// TwinCAT 3 PLC project PLC
// ProgramVersion: 3.1.4023.0
// libraries:
//   Tc2_EtherCAT, * (Beckhoff Automation GmbH)
//   Tc2_Standard, * (Beckhoff Automation GmbH)
//   Tc2_System, * (Beckhoff Automation GmbH)
//   Tc3_Module, * (Beckhoff Automation GmbH)
//   VisuDialogs, * (System)
// project tree:
//   / FastEL5131Task.TcTTO, GlobalTextList.TcGTLO, PlcTask.TcTTO, Visualization Manager.TcVMO (not stored)
//   POUs/ FB_PulseDiv.TcPOU, MAIN.TcPOU, MAINEL5131.TcPOU
//   VISUs/ MAINVISU.TcVIS
// real-time tasks:
//   TASK PlcTask: cycle T#10ms, priority 20, ADS port 350
//   TASK FastEL5131Task: cycle T#200us, priority 1, ADS port 351
// I/O:
//   DEVICE Device 1 (EtherCAT), AmsNetId 5.25.121.244.2.1
//     Term 1 (EK1100) [EK1100 EtherCAT Coupler (2A E-Bus)]
//       Term 2 (EL5131) [EL5131 1Ch. Inc. Encoder 5V (RS422,TTL), 2x24V DC Output]
//       Term 4 (EL5101) [EL5101 1Ch. Inc. Encoder 5V]
//       Term 3 (EL9011)
// variable links:
//   PLC Instance <-> Device 1 (EtherCAT)/Term 1 (EK1100)/Term 2 (EL5131)
//     FastEL5131Task Inputs/MAINEL5131.myPulseDiv.amsNetIdEL5131 <-> InfoData/AdsAddr/netId
//     FastEL5131Task Inputs/MAINEL5131.myPulseDiv.iEL5131CounterVal <-> ENC Status Channel 1/Counter value
//     FastEL5131Task Inputs/MAINEL5131.myPulseDiv.wPortEL5131 <-> InfoData/AdsAddr/port
//     FastEL5131Task Outputs/MAINEL5131.myPulseDiv.bEnbThreshOutputs <-> ENC Control Output Channel 1/Control Output/Control/Enable thresholds output
//     FastEL5131Task Outputs/MAINEL5131.myPulseDiv.bEnbThreshOutputs2 <-> ENC Control Output Channel 2/Control Output/Control/Enable thresholds output
//     FastEL5131Task Outputs/MAINEL5131.myPulseDiv.bForceResetCounter <-> ENC Control Channel 1/Control/Set counter
//     FastEL5131Task Outputs/MAINEL5131.myPulseDiv.bSetDigitalOut <-> ENC Control Output Channel 1/Control Output/Control/Set digital output
//     FastEL5131Task Outputs/MAINEL5131.myPulseDiv.bSetDigitalOut2 <-> ENC Control Output Channel 2/Control Output/Control/Set digital output
//     FastEL5131Task Outputs/MAINEL5131.myPulseDiv.iForceResetCntVal <-> ENC Control Channel 1/Set counter value
//     FastEL5131Task Outputs/MAINEL5131.myPulseDiv.iNbOfOutputEvents <-> ENC Control Output Channel 1/Control Output/Number of output events
//     FastEL5131Task Outputs/MAINEL5131.myPulseDiv.iOutStates_1[1] <-> ENC Control Output Channel 1/Control Output/Output state/Output state 1
//     FastEL5131Task Outputs/MAINEL5131.myPulseDiv.iOutStates_1[2] <-> ENC Control Output Channel 1/Control Output/Output state/Output state 2
//     FastEL5131Task Outputs/MAINEL5131.myPulseDiv.iOutStates_1[3] <-> ENC Control Output Channel 1/Control Output/Output state/Output state 3
//     FastEL5131Task Outputs/MAINEL5131.myPulseDiv.iOutStates_1[4] <-> ENC Control Output Channel 1/Control Output/Output state/Output state 4
//     FastEL5131Task Outputs/MAINEL5131.myPulseDiv.iOutStates_1[5] <-> ENC Control Output Channel 1/Control Output/Output state/Output state 5
//     FastEL5131Task Outputs/MAINEL5131.myPulseDiv.iOutStates_1[6] <-> ENC Control Output Channel 1/Control Output/Output state/Output state 6
//     FastEL5131Task Outputs/MAINEL5131.myPulseDiv.iOutStates_1[7] <-> ENC Control Output Channel 1/Control Output/Output state/Output state 7
//     FastEL5131Task Outputs/MAINEL5131.myPulseDiv.iOutStates_1[8] <-> ENC Control Output Channel 1/Control Output/Output state/Output state 8
//     FastEL5131Task Outputs/MAINEL5131.myPulseDiv.iOutStates_2[1] <-> ENC Control Output Channel 2/Control Output/Output state/Output state 1
//     FastEL5131Task Outputs/MAINEL5131.myPulseDiv.iOutStates_2[2] <-> ENC Control Output Channel 2/Control Output/Output state/Output state 2
//     FastEL5131Task Outputs/MAINEL5131.myPulseDiv.iOutStates_2[3] <-> ENC Control Output Channel 2/Control Output/Output state/Output state 3
//     FastEL5131Task Outputs/MAINEL5131.myPulseDiv.iOutStates_2[4] <-> ENC Control Output Channel 2/Control Output/Output state/Output state 4
//     FastEL5131Task Outputs/MAINEL5131.myPulseDiv.iOutStates_2[5] <-> ENC Control Output Channel 2/Control Output/Output state/Output state 5
//     FastEL5131Task Outputs/MAINEL5131.myPulseDiv.iOutStates_2[6] <-> ENC Control Output Channel 2/Control Output/Output state/Output state 6
//     FastEL5131Task Outputs/MAINEL5131.myPulseDiv.iOutStates_2[7] <-> ENC Control Output Channel 2/Control Output/Output state/Output state 7
//     FastEL5131Task Outputs/MAINEL5131.myPulseDiv.iOutStates_2[8] <-> ENC Control Output Channel 2/Control Output/Output state/Output state 8
//     FastEL5131Task Outputs/MAINEL5131.myPulseDiv.iThresholds_1 <-> ENC Control Output Channel 1/Control Output/Threshold/Threshold 1
//     FastEL5131Task Outputs/MAINEL5131.myPulseDiv.iThresholds_2 <-> ENC Control Output Channel 2/Control Output/Threshold/Threshold 1
//     FastEL5131Task Outputs/MAINEL5131.myPulseDiv.iThresholds_1 @bit 32 <-> ENC Control Output Channel 1/Control Output/Threshold/Threshold 2
//     FastEL5131Task Outputs/MAINEL5131.myPulseDiv.iThresholds_1 @bit 64 <-> ENC Control Output Channel 1/Control Output/Threshold/Threshold 3
//     FastEL5131Task Outputs/MAINEL5131.myPulseDiv.iThresholds_1 @bit 96 <-> ENC Control Output Channel 1/Control Output/Threshold/Threshold 4
//     FastEL5131Task Outputs/MAINEL5131.myPulseDiv.iThresholds_1 @bit 128 <-> ENC Control Output Channel 1/Control Output/Threshold/Threshold 5
//     FastEL5131Task Outputs/MAINEL5131.myPulseDiv.iThresholds_1 @bit 160 <-> ENC Control Output Channel 1/Control Output/Threshold/Threshold 6
//     FastEL5131Task Outputs/MAINEL5131.myPulseDiv.iThresholds_1 @bit 192 <-> ENC Control Output Channel 1/Control Output/Threshold/Threshold 7
//     FastEL5131Task Outputs/MAINEL5131.myPulseDiv.iThresholds_1 @bit 224 <-> ENC Control Output Channel 1/Control Output/Threshold/Threshold 8
//     FastEL5131Task Outputs/MAINEL5131.myPulseDiv.iThresholds_2 @bit 32 <-> ENC Control Output Channel 2/Control Output/Threshold/Threshold 2
//     FastEL5131Task Outputs/MAINEL5131.myPulseDiv.iThresholds_2 @bit 64 <-> ENC Control Output Channel 2/Control Output/Threshold/Threshold 3
//     FastEL5131Task Outputs/MAINEL5131.myPulseDiv.iThresholds_2 @bit 96 <-> ENC Control Output Channel 2/Control Output/Threshold/Threshold 4
//     FastEL5131Task Outputs/MAINEL5131.myPulseDiv.iThresholds_2 @bit 128 <-> ENC Control Output Channel 2/Control Output/Threshold/Threshold 5
//     FastEL5131Task Outputs/MAINEL5131.myPulseDiv.iThresholds_2 @bit 160 <-> ENC Control Output Channel 2/Control Output/Threshold/Threshold 6
//     FastEL5131Task Outputs/MAINEL5131.myPulseDiv.iThresholds_2 @bit 192 <-> ENC Control Output Channel 2/Control Output/Threshold/Threshold 7
//     FastEL5131Task Outputs/MAINEL5131.myPulseDiv.iThresholds_2 @bit 224 <-> ENC Control Output Channel 2/Control Output/Threshold/Threshold 8
//   PLC Instance <-> Device 1 (EtherCAT)/Term 1 (EK1100)/Term 4 (EL5101)
//     PlcTask Inputs/MAIN.iCounterValueDoubleCheckEL5101 <-> ENC Status/Counter value
//     PlcTask Outputs/MAIN.bResetCounterEL5101 <-> ENC Control/Control/Set counter
//     PlcTask Outputs/MAIN.iSetCounterValueEL5101ForReset <-> ENC Control/Set counter value

CONFIGURATION PLC
    RESOURCE PLC ON TwinCAT3
        TASK FastEL5131Task(INTERVAL := T#200us, PRIORITY := 1);
        TASK PlcTask(INTERVAL := T#10ms, PRIORITY := 20);
        PROGRAM MAINEL5131 WITH FastEL5131Task : MAINEL5131;
        PROGRAM MAIN WITH PlcTask : MAIN;
    END_RESOURCE
END_CONFIGURATION

// ---- POUs/MAINEL5131.TcPOU
PROGRAM MAINEL5131
VAR
	iDivRatio					:UINT:=4;
	iDivRatio2					:UINT:=5;
	iEvalMode					:USINT:=4;

	
	bSingleShot					:bool:=false;
	bReinitDivider				:BOOL;
	
	bDualMode					:BOOL;
	bFeed						:BOOL;
	
	trigReinitDivider			:r_trig;
END_VAR

END_PROGRAM

// ---- POUs/MAIN.TcPOU
PROGRAM MAIN
VAR
	iCounterValueDoubleCheckEL5101		AT%I*			:UDINT;
	bResetCounterEL5101					AT%Q*			:BOOL;
	iSetCounterValueEL5101ForReset		AT%Q*			:UDINT;
	
	bResetEL5101										:bool;
END_VAR

bResetCounterEL5101:=FALSE;

IF bResetEL5101 THEN
	bResetCounterEL5101:=TRUE;
	iSetCounterValueEL5101ForReset:=0;
	bResetEL5101:=FALSE;
END_IF

END_PROGRAM

// ---- POUs/FB_PulseDiv.TcPOU
FUNCTION_BLOCK FB_PulseDiv
VAR_INPUT
	///bSingleShotPulses=TRUE=> output pulses are as wide as 1/2 of the input pulses period
	bSingleShotPulses: BOOL;
	///bSingleShotPulses=FALS=> output pulses are generated with a 50% duty cyle
	iDividerRatio1stOutput: UINT;
	iDividerRatio2ndOutput: UINT;
	iEvalMode: USINT;
END_VAR
VAR_OUTPUT
	///this output is set to TRUE when the terminal has been configured
	bConfigured: BOOL;
END_VAR
VAR
	iEL5131CounterVal AT %I*: UDINT;
	iStatusDO1 AT %I*: BOOL;
	iStatusDO2 AT %I*: BOOL;
	///this variable controls the evolution of the configuration sequence
	stepCfgEL5131Single: USINT := 0;
	///info about error occurring while executing the config sequence of the EL5131
	bError: BOOL;
	///info about error occurring while executing the config sequence of the EL5131
	iErrStep: USINT;
	///identifying the correct EL5131 terminal
	amsNetIdEL5131 AT %I*: AMSNETID;
	sAmsNetIdEL5131: STRING;
	///identifying the correct EL5131 terminal
	wPortEL5131 AT %I*: WORD;
	///number of outputs events (always 2)	
	iNbOfOutputEvents AT %Q*: USINT;
	///for temporarily disabling the writing of the output based on counter thresholds, while reconfiguring the terminal 
	bEnbThreshOutputs AT %Q*: BOOL;
	///for temporarily disabling the writing of the output based on counter thresholds, while reconfiguring the terminal 
	bEnbThreshOutputs2 AT %Q*: BOOL;
	///for temporarily  forcing the output to FALSE, while reconfiguring the terminal
	bSetDigitalOut AT %Q*: BOOL;
	///for temporarily  forcing the output to FALSE, while reconfiguring the terminal
	bSetDigitalOut2 AT %Q*: BOOL;
	///value for the output_1 thresholds, 
	iThresholds_1 AT %Q*: ARRAY[1..8] OF UDINT;
	///output_1 events
	iOutStates_1 AT %Q*: ARRAY[1..8] OF BOOL;
	///value for the output_2 thresholds, 
	iThresholds_2 AT %Q*: ARRAY[1..8] OF UDINT;
	///output_2 events
	iOutStates_2 AT %Q*: ARRAY[1..8] OF BOOL;
	///force reset the counter value to 0 when the EL5131 is reconfigured
	bForceResetCounter AT %Q*: BOOL;
	///force reset the counter value to 0 when the EL5131 is reconfigured
	iForceResetCntVal AT %Q*: UDINT;
	arrFIFO_Thr_1: ARRAY[1..20] OF UDINT;
	arrFIFO_Evt_1: ARRAY[1..20] OF BOOL;
	arrFIFO_Thr_2: ARRAY[1..20] OF UDINT;
	arrFIFO_Evt_2: ARRAY[1..20] OF BOOL;
	///in order to be able to overwrite the limit counter value and reset counter value via CoE in the EL5131, the value 16#72657375 needs to be written in the object 16#F008 
	iProtectionReg: UDINT := 16#72657375;
	///defining the max limit counter value at which the counter is automatically reset to the reset counter value
	iLimitCounterVal: UDINT := 31;
	///start value of the counter once it has been reset	
	iResetCounterVal: UDINT := 0;
	writeCoEConfig: FB_EcCoESdoWrite;
	///Evaluation mode (1-fold, 2-fold, 4-fold) is chosen via a Property of the FB; Divider ratio (4,5,7) is chosen via a Property of the FB
	iSelectedEvalMode: USINT;
	iCoeEnumEvalMode: USINT;
	iDividerRatio: UINT;
	///Dual mode
	stepCfgEL5131Dual: USINT := 0;
	///only in dual output mode
	iDividerRatio2: UINT;
	iNbOfOutputEvents2 AT %Q*: USINT;
	iCntLimDivider: UDINT;
	iCntLimDivider2: UDINT;
	iCntLimDividerMin: UDINT;
	iDualCntLimit: UDINT;
	iHalfOutPeriodNrOfEvts: UDINT;
	iHalfOutPeriodNrOfEvts2: UDINT;
	iNumberOfEventsCycle: UDINT;
	iNumberOfEventsCycle2: UDINT;
	idx: UDINT;
	iArr: UINT;
	i: UINT;
	j: UINT;
	iGcd: UDINT;
	///Fifo feed when Dual outputs are used
	idxFeed: UDINT;
	idxFIFO: UDINT;
END_VAR

sAmsNetIdEL5131:=F_CreateAmsNetId(amsNetIdEL5131);

writeCoEConfig(
	sNetId:=sAmsNetIdEL5131 , 
	nSlaveAddr:=wPortEL5131 , 
	nSubIndex:= , 
	nIndex:= , 
	pSrcBuf:= , 
	cbBufLen:= , 
	bExecute:= , 
	tTimeout:=T#3S , 
	bBusy=> , 
	bError=> , 
	nErrId=> );
	
iDividerRatio:=LIMIT(2,iDividerRatio1stOutput,20);	
iDividerRatio2:=LIMIT(2,iDividerRatio2ndOutput,20);	
	

IF ((iEvalMode<>1) AND (iEvalMode<>2) AND (iEvalMode<>4)) THEN
	iSelectedEvalMode:=4;  //iEvaluationMode=4 =>Quadrature decoding
ELSE
	iSelectedEvalMode:=iEvalMode;
END_IF
		
CASE iSelectedEvalMode OF
	1: iCoeEnumEvalMode:=1; (*1-fold*)
	2: iCoeEnumEvalMode:=2; (*2-fold*)
	4: iCoeEnumEvalMode:=0; (*4-fold*)		
END_CASE

	
//triggering the start of the sequence, when the Method is explicitly called
IF stepCfgEL5131Single=0 THEN
	bConfigured:=FALSE;
	iErrStep:=0;
	bError:=FALSE;
	stepCfgEL5131Single:=1;
END_IF

/////////////////////////////////////////////////////////////////////////////////////////////////////////////////////////////////////////////////////////////////
///////////////////////////////////////////////////SEQUENCE FOR INITIALIZING A SINGLE PULSE TRAIN DIVIDER OUTPUT/////////////////////////////////////////////////
/////////////////////////////////////////////////////////////////////////////////////////////////////////////////////////////////////////////////////////////////
//step sequence for the different configuration steps of the EL5131
CASE stepCfgEL5131Single OF
	
	//disabling the output threshold comparison/activation so the output can be forced to FALSE in the next step
	1: 	bEnbThreshOutputs:=FALSE;
		bEnbThreshOutputs2:=FALSE;
		stepCfgEL5131Single:=2;
		
	//forcing the output to FALSE, so the output pulse train will start with a 0 level, after the EL5131 has been reconfigured
	2:	bSetDigitalOut:=FALSE;
		bSetDigitalOut2:=FALSE;
		stepCfgEL5131Single:=3;
		
	//resetting the counter of the EL5131 to the value 0, so the terminal will start counting from the very first puls after it has been reconfigured
	3:	iForceResetCntVal:=0;
		bForceResetCounter:=TRUE;
		stepCfgEL5131Single:=4;
		
	//re-activating the output activation on the basis of counter thresholds comparison	
	4:	bForceResetCounter:=FALSE;
		bEnbThreshOutputs:=TRUE;
		stepCfgEL5131Single:=10;

	
	//prepare values for pulse divider 
	10:	iNbOfOutputEvents:=2;	
		iNbOfOutputEvents2:=0;
		iResetCounterVal:=0;	//the encoder counter value is always counting starting from 0

		IF bSingleShotPulses THEN	//here is chosen if the output pulse train will be a 50% duty cycle wave of single-shot pulses		
			iLimitCounterVal:=iSelectedEvalMode*iDividerRatio-1;	//the encoder value counts up to iLimitCounterVal then is automatically reset to iResetCounterVal internally in the terminal
			
			iThresholds_1[1]:=iSelectedEvalMode*iDividerRatio-1;	
			iOutStates_1[1]:=TRUE;
			
			iThresholds_1[2]:=0;
			iOutStates_1[2]:=FALSE;			
		ELSE
			iLimitCounterVal:=iSelectedEvalMode*iDividerRatio-1;	//the encoder value counts up to iLimitCounterVal then is automatically reset to iResetCounterVal internally in the terminal
			
			iThresholds_1[1]:=iSelectedEvalMode*iDividerRatio/2;	//old (iSelectedEvalMode*iDividerRatio/2)-1
			iOutStates_1[1]:=TRUE;
			
			iThresholds_1[2]:=0;									// old iSelectedEvalMode*iDividerRatio-1;
			iOutStates_1[2]:=FALSE;		
		END_IF;	
	
			stepCfgEL5131Single:=20;

	//write ascii USER into register 0xF008 to lift protection on counter reset/limit values in the terminal
	//this has to be done if the CoE objects 16#8001:1A (limit counter value) and 16#8001:1B (reset counter value);	
	20:	iProtectionReg:=16#72657375;
		writeCoEConfig.nIndex:=16#F008;
		writeCoEConfig.nSubIndex:=16#00;
		writeCoEConfig.pSrcBuf:=ADR(iProtectionReg);
		writeCoEConfig.cbBufLen:=SIZEOF(iProtectionReg);
		
		writeCoEConfig.bExecute:=TRUE;
		
		IF writeCoEConfig.bBusy THEN
			writeCoEConfig.bExecute:=FALSE;
			stepCfgEL5131Single:=30;
		END_IF;
		
	//wait for the end of writing the limit counter value	
	30: IF NOT writeCoEConfig.bBusy AND NOT writeCoEConfig.bError THEN
			stepCfgEL5131Single:=40;			
		END_IF
		
		IF writeCoEConfig.bError THEN
			bError:=TRUE;
			iErrStep:=stepCfgEL5131Single;
			stepCfgEL5131Single:=0;
		END_IF


	//write limit counter value	= max value of the counter from which the EL5131 terminal restarts counting from the reset counter value	
	40:	writeCoEConfig.nIndex:=16#8001;
		writeCoEConfig.nSubIndex:=16#1A;
		writeCoEConfig.pSrcBuf:=ADR(iLimitCounterVal);
		writeCoEConfig.cbBufLen:=SIZEOF(iLimitCounterVal);
		
		writeCoEConfig.bExecute:=TRUE;
		
		IF writeCoEConfig.bBusy THEN
			writeCoEConfig.bExecute:=FALSE;
			stepCfgEL5131Single:=50;
		END_IF;
		
	//wait for the end of writing the limit counter value	
	50: IF NOT writeCoEConfig.bBusy AND NOT writeCoEConfig.bError THEN
			stepCfgEL5131Single:=60;			
		END_IF
		
		IF writeCoEConfig.bError THEN
			bError:=TRUE;
			iErrStep:=stepCfgEL5131Single;
			stepCfgEL5131Single:=0;
		END_IF

	//write reset counter value	= starting value for the counter whe it is reset (normally 0)	
	60:	writeCoEConfig.nIndex:=16#8001;
		writeCoEConfig.nSubIndex:=16#1B;
		writeCoEConfig.pSrcBuf:=ADR(iResetCounterVal);
		writeCoEConfig.cbBufLen:=SIZEOF(iResetCounterVal);
		
		writeCoEConfig.bExecute:=TRUE;
		
		IF writeCoEConfig.bBusy THEN
			writeCoEConfig.bExecute:=FALSE;
			stepCfgEL5131Single:=70;
		END_IF;
		
	//wait for the end of writing the reset counter value	
	70: IF NOT writeCoEConfig.bBusy AND NOT writeCoEConfig.bError THEN
			stepCfgEL5131Single:=80;			
		END_IF
		
		IF writeCoEConfig.bError THEN
			bError:=TRUE;
			iErrStep:=stepCfgEL5131Single;
			stepCfgEL5131Single:=0;
		END_IF
		
	//write the evaluation mode: 1-fold, (value 1)  2-fold (value 2) or 4-fold (value 0)	
	//1-fold = only the rising edges of the encoder A-track are counted	
	//2-fold = both the rising and falling edges of the encoder A-track are counted	
	//4-fold = both the rising and falling edges of the encoder A and B tracks are counted	
	80:	writeCoEConfig.nIndex:=16#8000;
		writeCoEConfig.nSubIndex:=16#06;
		writeCoEConfig.pSrcBuf:=ADR(iCoeEnumEvalMode);
		writeCoEConfig.cbBufLen:=SIZEOF(iCoeEnumEvalMode);
		
		writeCoEConfig.bExecute:=TRUE;
		
		IF writeCoEConfig.bBusy THEN
			writeCoEConfig.bExecute:=FALSE;
			stepCfgEL5131Single:=90;
		END_IF;
		
	//wait for the end of writing the evaluation mode	
	90: IF NOT writeCoEConfig.bBusy AND NOT writeCoEConfig.bError THEN
			stepCfgEL5131Single:=100;			
		END_IF
		
		IF writeCoEConfig.bError THEN
			bError:=TRUE;
			iErrStep:=stepCfgEL5131Single;
			stepCfgEL5131Single:=0;
		END_IF		
	
	//write 0 into register 0xF008 to set protection on counter reset/limit values, after they have been changed earlier in the sequence	
	100:iProtectionReg:=16#00000000;
		writeCoEConfig.nIndex:=16#F008;
		writeCoEConfig.nSubIndex:=16#00;
		writeCoEConfig.pSrcBuf:=ADR(iProtectionReg);
		writeCoEConfig.cbBufLen:=SIZEOF(iProtectionReg);
		
		writeCoEConfig.bExecute:=TRUE;
		
		IF writeCoEConfig.bBusy THEN
			writeCoEConfig.bExecute:=FALSE;
			stepCfgEL5131Single:=110;
		END_IF;
		
	//wait for the end of writing 	
	110: IF NOT writeCoEConfig.bBusy AND NOT writeCoEConfig.bError THEN
			bConfigured:=TRUE;	//setting the 'bConfigured' bit so it is confirmed that the sequence has been completely executed
			stepCfgEL5131Single:=0;			
		END_IF
		
		IF writeCoEConfig.bError THEN
			bError:=TRUE;
			iErrStep:=stepCfgEL5131Single;
			stepCfgEL5131Single:=0;
		END_IF
	
		
END_CASE
/////////////////////////////////////////////////////////////////////////////////////////////////////////////////////////////////////////////////////////////////
///////////////////////////////////////////////////SEQUENCE FOR INITIALIZING A SINGLE PULSE TRAIN DIVIDER OUTPUT/////////////////////////////////////////////////
/////////////////////////////////////////////////////////////////////////////////////////////////////////////////////////////////////////////////////////////////



/////////////////////////////////////////////////////////////////////////////////////////////////////////////////////////////////////////////////////////////////
/////////////////////////////////////////////////////SEQUENCE FOR INITIALIZING A DUAL PULSE TRAIN DIVIDER OUTPUT/////////////////////////////////////////////////
/////////////////////////////////////////////////////////////////////////////////////////////////////////////////////////////////////////////////////////////////
//triggering the start of the sequence, when the Method is explicitly called
IF stepCfgEL5131Dual=0 THEN
	bConfigured:=FALSE;
	iErrStep:=0;
	bError:=FALSE;
	stepCfgEL5131Dual:=1;
END_IF


//step sequence for the different configuration steps of the EL5131
CASE stepCfgEL5131Dual OF
	
	//disabling the output threshold comparison/activation so the output can be forced to FALSE in the next step
	1: 	bEnbThreshOutputs:=FALSE;
		bEnbThreshOutputs2:=FALSE;
		stepCfgEL5131Dual:=2;
		
	//forcing the output to FALSE, so the output pulse train will start with a 0 level, after the EL5131 has been reconfigured
	2:	bSetDigitalOut:=FALSE;
		bSetDigitalOut2:=FALSE;
		stepCfgEL5131Dual:=3;
		
	//resetting the counter of the EL5131 to the value 0, so the terminal will start counting from the very first puls after it has been reconfigured
	3:	iForceResetCntVal:=0;
		bForceResetCounter:=TRUE;
		stepCfgEL5131Dual:=4;
		
	//re-activating the output activation on the basis of counter thresholds comparison	
	4:	bForceResetCounter:=FALSE;
		bEnbThreshOutputs:=TRUE;
		bEnbThreshOutputs2:=TRUE;
		stepCfgEL5131Dual:=5;
		
	//calculating the least common multiple of both counter limits	
	5: 	iCntLimDivider:=iSelectedEvalMode*iDividerRatio;
		iCntLimDivider2:=iSelectedEvalMode*iDividerRatio2;
		
		iCntLimDividerMin:=MIN(iCntLimDivider,iCntLimDivider2);
		
		//first searching the greatest common divisor=the biggest number that commonly divides both counters, without remainder
		FOR idx:=1 TO iCntLimDivider DO
			IF (iCntLimDivider MOD idx=0) AND (iCntLimDivider2 MOD idx=0) THEN
				iGcd:=idx;
			END_IF
		END_FOR		
		
		//now that we have the greatest common divisor, we can calculate the least common multiple
		IF iGcd<>0 THEN	
			iDualCntLimit:=iCntLimDivider*iCntLimDivider2/iGcd;
			stepCfgEL5131Dual:=10;
		ELSE
			iDualCntLimit:=0;
			stepCfgEL5131Dual:=0;
			iErrStep:=5;
			bError:=TRUE;
		END_IF;
			
	//prepare values for pulse divider 
	10:	iLimitCounterVal:=iDualCntLimit-1;	//the encoder value counts up to iLimitCounterVal then is automatically reset to iResetCounterVal internally in the terminal
		iResetCounterVal:=0;	//the encoder counter value is always counting starting from 0			
	
		iHalfOutPeriodNrOfEvts:=(iSelectedEvalMode*iDividerRatio)/2;
		iHalfOutPeriodNrOfEvts2:=(iSelectedEvalMode*iDividerRatio2)/2;		
		
		IF (iHalfOutPeriodNrOfEvts>0) THEN
			iNumberOfEventsCycle:=(iDualCntLimit/iHalfOutPeriodNrOfEvts);
		END_IF;
	
		IF (iHalfOutPeriodNrOfEvts2>0) THEN
			iNumberOfEventsCycle2:=(iDualCntLimit/iHalfOutPeriodNrOfEvts2);
		END_IF;
			
		FOR idx:=1 TO 20 DO
			arrFIFO_Thr_1[idx]:=0;
			arrFIFO_Evt_1[idx]:=0;
			arrFIFO_Thr_2[idx]:=0;
			arrFIFO_Evt_2[idx]:=0;
		END_FOR
		
		FOR idx:=1 TO iNumberOfEventsCycle DO
			arrFIFO_Thr_1[idx]:=iHalfOutPeriodNrOfEvts*(idx-1); 
			arrFIFO_Evt_1[idx]:=(idx MOD 2=0);	
		END_FOR
	
		FOR idx:=1 TO iNumberOfEventsCycle2 DO
			arrFIFO_Thr_2[idx]:=iHalfOutPeriodNrOfEvts2*(idx-1); 
			arrFIFO_Evt_2[idx]:=(idx MOD 2=0);	
		END_FOR
		
		iNbOfOutputEvents:=LIMIT(0,TO_USINT(iNumberOfEventsCycle),8);	
		iNbOfOutputEvents2:=Limit(0,TO_USINT(iNumberOfEventsCycle2),8);	
	
		stepCfgEL5131Dual:=20;

	//write ascii USER into register 0xF008 to lift protection on counter reset/limit values in the terminal
	//this has to be done if the CoE objects 16#8001:1A (limit counter value) and 16#8001:1B (reset counter value);	
	20:	iProtectionReg:=16#72657375;
		writeCoEConfig.nIndex:=16#F008;
		writeCoEConfig.nSubIndex:=16#00;
		writeCoEConfig.pSrcBuf:=ADR(iProtectionReg);
		writeCoEConfig.cbBufLen:=SIZEOF(iProtectionReg);
		
		writeCoEConfig.bExecute:=TRUE;
		
		IF writeCoEConfig.bBusy THEN
			writeCoEConfig.bExecute:=FALSE;
			stepCfgEL5131Dual:=30;
		END_IF;
		
	//wait for the end of writing the limit counter value	
	30: IF NOT writeCoEConfig.bBusy AND NOT writeCoEConfig.bError THEN
			stepCfgEL5131Dual:=40;			
		END_IF
		
		IF writeCoEConfig.bError THEN
			bError:=TRUE;
			iErrStep:=stepCfgEL5131Dual;
			stepCfgEL5131Dual:=0;
		END_IF


	//write limit counter value	= max value of the counter from which the EL5131 terminal restarts counting from the reset counter value	
	40:	writeCoEConfig.nIndex:=16#8001;
		writeCoEConfig.nSubIndex:=16#1A;
		writeCoEConfig.pSrcBuf:=ADR(iLimitCounterVal);
		writeCoEConfig.cbBufLen:=SIZEOF(iLimitCounterVal);
		
		writeCoEConfig.bExecute:=TRUE;
		
		IF writeCoEConfig.bBusy THEN
			writeCoEConfig.bExecute:=FALSE;
			stepCfgEL5131Dual:=50;
		END_IF;
		
	//wait for the end of writing the limit counter value	
	50: IF NOT writeCoEConfig.bBusy AND NOT writeCoEConfig.bError THEN
			stepCfgEL5131Dual:=60;			
		END_IF
		
		IF writeCoEConfig.bError THEN
			bError:=TRUE;
			iErrStep:=stepCfgEL5131Dual;
			stepCfgEL5131Dual:=0;
		END_IF

	//write reset counter value	= starting value for the counter whe it is reset (normally 0)	
	60:	writeCoEConfig.nIndex:=16#8001;
		writeCoEConfig.nSubIndex:=16#1B;
		writeCoEConfig.pSrcBuf:=ADR(iResetCounterVal);
		writeCoEConfig.cbBufLen:=SIZEOF(iResetCounterVal);
		
		writeCoEConfig.bExecute:=TRUE;
		
		IF writeCoEConfig.bBusy THEN
			writeCoEConfig.bExecute:=FALSE;
			stepCfgEL5131Dual:=70;
		END_IF;
		
	//wait for the end of writing the reset counter value	
	70: IF NOT writeCoEConfig.bBusy AND NOT writeCoEConfig.bError THEN
			stepCfgEL5131Dual:=80;			
		END_IF
		
		IF writeCoEConfig.bError THEN
			bError:=TRUE;
			iErrStep:=stepCfgEL5131Dual;
			stepCfgEL5131Dual:=0;
		END_IF
		
	//write the evaluation mode: 1-fold, (value 1)  2-fold (value 2) or 4-fold (value 0)	
	//1-fold = only the rising edges of the encoder A-track are counted	
	//2-fold = both the rising and falling edges of the encoder A-track are counted	
	//4-fold = both the rising and falling edges of the encoder A and B tracks are counted	
	80:	writeCoEConfig.nIndex:=16#8000;
		writeCoEConfig.nSubIndex:=16#06;
		writeCoEConfig.pSrcBuf:=ADR(iCoeEnumEvalMode);
		writeCoEConfig.cbBufLen:=SIZEOF(iCoeEnumEvalMode);
		
		writeCoEConfig.bExecute:=TRUE;
		
		IF writeCoEConfig.bBusy THEN
			writeCoEConfig.bExecute:=FALSE;
			stepCfgEL5131Dual:=90;
		END_IF;
		
	//wait for the end of writing the evaluation mode	
	90: IF NOT writeCoEConfig.bBusy AND NOT writeCoEConfig.bError THEN
			stepCfgEL5131Dual:=100;			
		END_IF
		
		IF writeCoEConfig.bError THEN
			bError:=TRUE;
			iErrStep:=stepCfgEL5131Dual;
			stepCfgEL5131Dual:=0;
		END_IF		
	
	//write 0 into register 0xF008 to set protection on counter reset/limit values, after they have been changed earlier in the sequence	
	100:iProtectionReg:=16#00000000;
		writeCoEConfig.nIndex:=16#F008;
		writeCoEConfig.nSubIndex:=16#00;
		writeCoEConfig.pSrcBuf:=ADR(iProtectionReg);
		writeCoEConfig.cbBufLen:=SIZEOF(iProtectionReg);
		
		writeCoEConfig.bExecute:=TRUE;
		
		IF writeCoEConfig.bBusy THEN
			writeCoEConfig.bExecute:=FALSE;
			stepCfgEL5131Dual:=110;
		END_IF;
		
	//wait for the end of writing 	
	110: IF NOT writeCoEConfig.bBusy AND NOT writeCoEConfig.bError THEN
			bConfigured:=TRUE;	//setting the 'bConfigured' bit so it is confirmed that the sequence has been completely executed
			stepCfgEL5131Dual:=0;			
		END_IF
		
		IF writeCoEConfig.bError THEN
			bError:=TRUE;
			iErrStep:=stepCfgEL5131Dual;
			stepCfgEL5131Dual:=0;
		END_IF
	
		
END_CASE
/////////////////////////////////////////////////////////////////////////////////////////////////////////////////////////////////////////////////////////////////
/////////////////////////////////////////////////////SEQUENCE FOR INITIALIZING A DUAL PULSE TRAIN DIVIDER OUTPUT/////////////////////////////////////////////////
/////////////////////////////////////////////////////////////////////////////////////////////////////////////////////////////////////////////////////////////////


/////////////////////////////////////////////////////////////////////////////////////////////////////////////////////////////////////////////////////////////////
///////////////////////////////////////////////////////////////////FIFO FEED WHEN DUAL OUTPUTS ARE USED//////////////////////////////////////////////////////////
/////////////////////////////////////////////////////////////////////////////////////////////////////////////////////////////////////////////////////////////////
//FIRST PULSE TRAIN/////////////////////////////////////////////////////////////////////////
//checking if we have more than 8 events/cycle; if not=>fixed counters; if yes=>FIFO feed 
IF iNumberOfEventsCycle<=8 THEN
	FOR idxFeed:=1 TO iNumberOfEventsCycle DO
		iThresholds_1[idxFeed]:=arrFIFO_Thr_1[idxFeed];
		iOutStates_1[idxFeed]:=arrFIFO_Evt_1[idxFeed];
	END_FOR
ELSE	
	//search the next FIFO value the closest to the actual counter value
	idxFifo:=1;
	FOR idxFeed:=1 TO iNumberOfEventsCycle DO
		IF iThresholds_1[idxFeed]>=iEL5131CounterVal THEN
			idxFIFO:=idxFeed;
			EXIT;
		END_IF;
	END_FOR;	
	FOR idxFeed:=1 TO 8 DO
		IF (idxFIFO+idxFeed-1)<=iNumberOfEventsCycle THEN
			iThresholds_1[idxFeed]:=arrFIFO_Thr_1[idxFIFO+idxFeed-1];
			iOutStates_1[idxFeed]:=arrFIFO_Evt_1[idxFIFO+idxFeed-1];	
		ELSE
			iThresholds_1[idxFeed]:=arrFIFO_Thr_1[idxFIFO+idxFeed-1-iNumberOfEventsCycle];
			iOutStates_1[idxFeed]:=arrFIFO_Evt_1[idxFIFO+idxFeed-1-iNumberOfEventsCycle];				
		END_IF;	
	END_FOR

END_IF		
//////////////////////////////////////////////////////////////////////////////////////////////





//SECOND PULSE TRAIN/////////////////////////////////////////////////////////////////////////
//checking if we have more than 8 events/cycle; if not=>fixed counters; if yes=>FIFO feed 
IF iNumberOfEventsCycle2<=8 THEN
	FOR idxFeed:=1 TO iNumberOfEventsCycle2 DO
		iThresholds_2[idxFeed]:=arrFIFO_Thr_2[idxFeed];
		iOutStates_2[idxFeed]:=arrFIFO_Evt_2[idxFeed];
	END_FOR
ELSE	
	//search the next FIFO value the closest to the actual counter value
	idxFifo:=1;
	FOR idxFeed:=1 TO iNumberOfEventsCycle2 DO
		IF iThresholds_2[idxFeed]>=iEL5131CounterVal THEN
			idxFIFO:=idxFeed;
			EXIT;
		END_IF;
	END_FOR;	
	FOR idxFeed:=1 TO 8 DO
		IF (idxFIFO+idxFeed-1)<=iNumberOfEventsCycle2 THEN
			iThresholds_2[idxFeed]:=arrFIFO_Thr_2[idxFIFO+idxFeed-1];
			iOutStates_2[idxFeed]:=arrFIFO_Evt_2[idxFIFO+idxFeed-1];	
		ELSE
			iThresholds_2[idxFeed]:=arrFIFO_Thr_2[idxFIFO+idxFeed-1-iNumberOfEventsCycle2];
			iOutStates_2[idxFeed]:=arrFIFO_Evt_2[idxFIFO+idxFeed-1-iNumberOfEventsCycle2];				
		END_IF;	
	END_FOR

END_IF		
//////////////////////////////////////////////////////////////////////////////////////////////
/////////////////////////////////////////////////////////////////////////////////////////////////////////////////////////////////////////////////////////////////
///////////////////////////////////////////////////////////////////FIFO FEED WHEN DUAL OUTPUTS ARE USED//////////////////////////////////////////////////////////
/////////////////////////////////////////////////////////////////////////////////////////////////////////////////////////////////////////////////////////////////

END_FUNCTION_BLOCK

// ---- GlobalTextList.TcGTLO
TEXTLIST GlobalTextList
  504 = ' Counter actual value: %i'
  559 = ' EL5101'
  228 = ' EL5131'
  179 = ' Pulse train divider ratio 2: %i'
  384 = ' Pulse train divider ratio: %i'
  537 = ' x-fold evaluation: %i'
  107 = 'Counting generated pulses \n@output EL5131'
  338 = 'Counting generated pulses @output EL5131'
  430 = 'Dual mode'
  458 = 'EL5101'
  838 = 'EL5131'
  128 = 'Encoder '
  452 = 'Encoder analysis and\npulse train generator'
  131 = 'Pulse train divider ratio'
  819 = 'Pulse train divider ratio: %i'
  390 = 'Re-configure EL5131'
  423 = 'Reset counter EL5101'
  967 = 'Single-shot pulses'
END_TEXTLIST

// ---- VISUs/MAINVISU.TcVIS
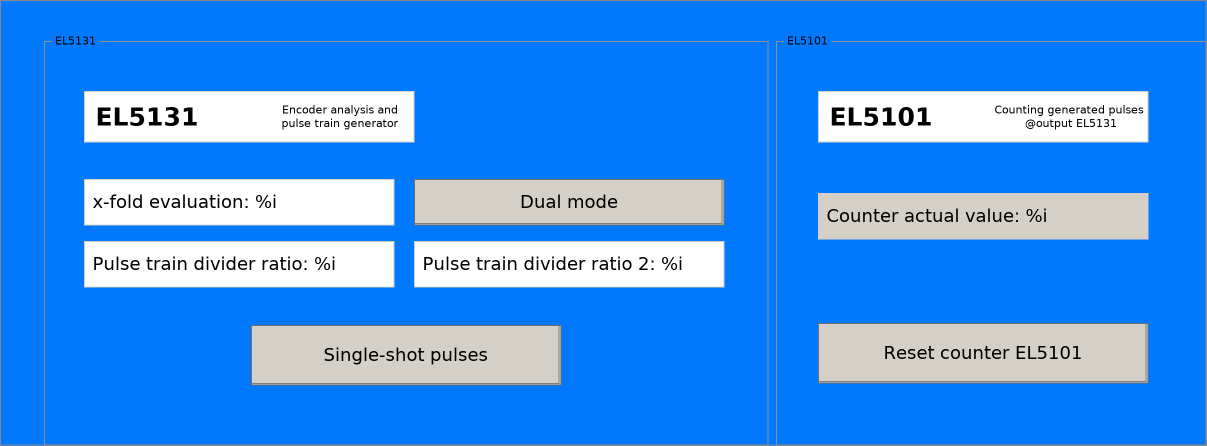
VISUALIZATION MAINVISU  // 1207x446
    GroupBox (44,33 724x413), "EL5131"
        Textfield (370,208 310x46), "Pulse train divider ratio 2: %i", text variable: MAINEL5131.iDivRatio2, invisible if: not MAINEL5131.bDualMode
            OnMouseClick: write the text variable via VisuDialogs.Numpad, min 2, max 20
        Button (370,146 310x46), "Dual mode"
            toggle MAINEL5131.bDualMode
        Textfield (40,146 310x46), "x-fold evaluation: %i", text variable: MAINEL5131.iEvalMode
            OnMouseClick: write the text variable via VisuDialogs.Numpad, min 1, max 4
        Button (207,292 310x60), "Single-shot pulses"
            toggle MAINEL5131.bSingleShot
    Textfield (84,91 330x51), "EL5131"
    Textfield (84,241 310x46), "Pulse train divider ratio: %i", text variable: MAINEL5131.iDivRatio
        OnMouseClick: write the text variable via VisuDialogs.Numpad, min 2, max 20
    Label (262,95 156x43), "Encoder analysis and pulse train generator"
    GroupBox (776,33 431x413), "EL5101"
    Textfield (818,91 330x51), "EL5101"
    Textfield (818,193 330x46), "Counter actual value: %i", text variable: MAIN.iCounterValueDoubleCheckEL5101
    Button (818,323 330x60), "Reset counter EL5101"
        tap MAIN.bResetEL5101
    Label (993,95 156x43), "Counting generated pulses @output EL5131"
END_VISUALIZATION
